(* Schneider Machine Expert - Basic project SEMÁFORO 1 VIA - SCHNEIDER ELECTRIC, file version 2.8.0.0 *)
(* ProjectInformations: Name=SEMAFORO 1 VIA, Description=Semáforo de 1 via com temporizadores., botão [LIGA], botão [DESLIGA] e repetição automática de ciclo. *)
(* UserInformations: LastName=Gagliano, FirstName=Leonardo *)

HARDWARE
  Cpu 0: TM221C40T
  EthernetConfiguration: NetworkName=M221, IpAllocationMode=FixedAddress, IpAddress=0.0.0.0, SubnetMask=0.0.0.0
  SerialLineConfiguration: Baud=Baud19200, Parity=ParityEven, DataBits=DataBits8, StopBits=StopBits1, PhysicalMedium=PhysicalMediumRs485, TransmissionMode=TransmissionModeModbusRtu, SlaveId=1, Addressing=SlaveAddressing
  MastTask: UsePeriodScanMode=false, PeriodScan=100
  FastTask: Period=255
  CpuBehavior: StartingMode=StartAsPreviousState, AutoSaveRamOnEeprom=true, WatchdogPeriod=250

SYMBOLS  (address, symbol, comment, settings)
  %M0       DESLIGA
  %TM0        [Preset=7, Base=OneSecond]
  %TM1        [Preset=3, Base=OneSecond]
  %TM2        [Preset=5, Base=OneSecond]
  %I0.0     LIGA
  %Q0.0     LUZ_VERMELHA
  %Q0.1     LUZ_AMARELA
  %Q0.2     LUZ_VERDE

POU Novo POU
  (* SectionNumber=1 *)

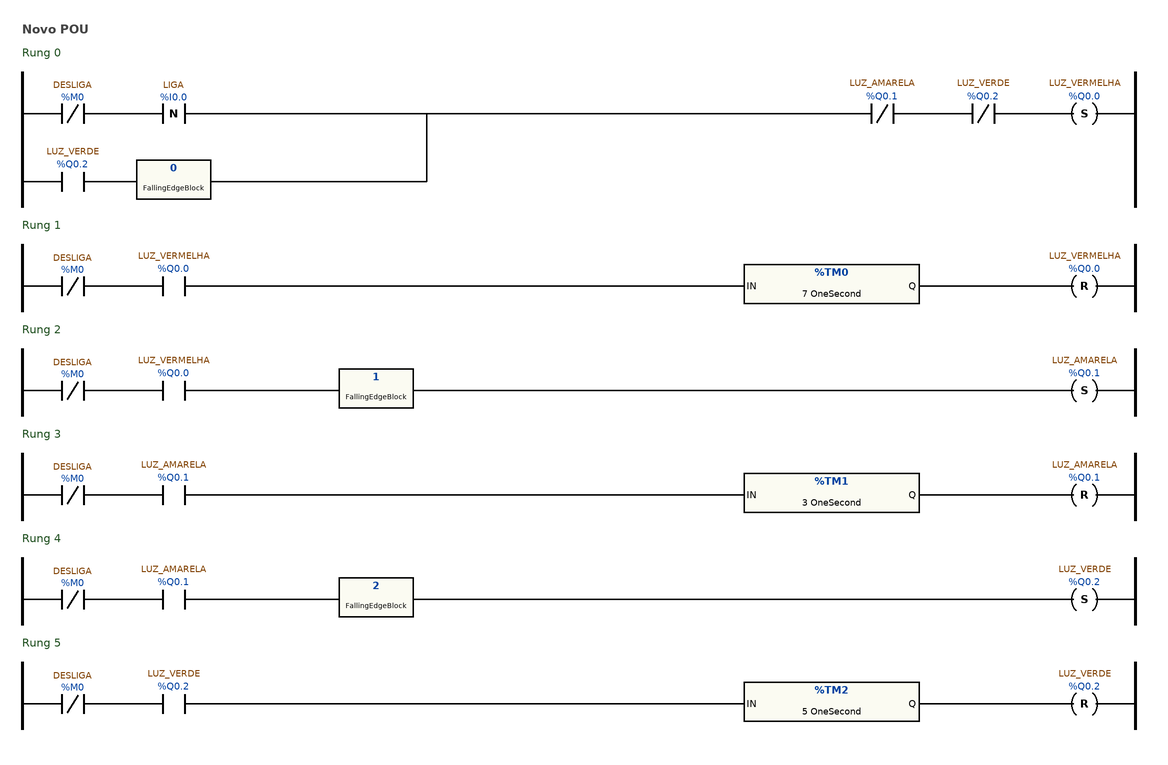

// Rung 0
  LDN %M0                 (* DESLIGA *)
  ANDF %I0.0              (* LIGA *)
  OR( %Q0.2               (* LUZ_VERDE *)
  FALLING0
  )
  ANDN %Q0.1              (* LUZ_AMARELA *)
  ANDN %Q0.2              (* LUZ_VERDE *)
  S %Q0.0                 (* LUZ_VERMELHA *)
  // as ST:
  //   IF (NOT DESLIGA AND FALLING(LIGA) OR FALLING(LUZ_VERDE)) AND NOT LUZ_AMARELA AND NOT LUZ_VERDE THEN LUZ_VERMELHA := TRUE; END_IF;

// Rung 1
  BLK %TM0
  LDN %M0                 (* DESLIGA *)
  AND %Q0.0               (* LUZ_VERMELHA *)
  IN
  OUT_BLK
  LD Q
  R %Q0.0                 (* LUZ_VERMELHA *)
  END_BLK
  // as ST:
  //   %TM0(IN := NOT DESLIGA AND LUZ_VERMELHA);
  //   IF %TM0.Q THEN LUZ_VERMELHA := FALSE; END_IF;

// Rung 2
  LDN %M0                 (* DESLIGA *)
  AND %Q0.0               (* LUZ_VERMELHA *)
  FALLING3
  S %Q0.1                 (* LUZ_AMARELA *)
  // as ST:
  //   IF FALLING(NOT DESLIGA AND LUZ_VERMELHA) THEN LUZ_AMARELA := TRUE; END_IF;

// Rung 3
  BLK %TM1
  LDN %M0                 (* DESLIGA *)
  AND %Q0.1               (* LUZ_AMARELA *)
  IN
  OUT_BLK
  LD Q
  R %Q0.1                 (* LUZ_AMARELA *)
  END_BLK
  // as ST:
  //   %TM1(IN := NOT DESLIGA AND LUZ_AMARELA);
  //   IF %TM1.Q THEN LUZ_AMARELA := FALSE; END_IF;

// Rung 4
  LDN %M0                 (* DESLIGA *)
  AND %Q0.1               (* LUZ_AMARELA *)
  FALLING2
  S %Q0.2                 (* LUZ_VERDE *)
  // as ST:
  //   IF FALLING(NOT DESLIGA AND LUZ_AMARELA) THEN LUZ_VERDE := TRUE; END_IF;

// Rung 5
  BLK %TM2
  LDN %M0                 (* DESLIGA *)
  AND %Q0.2               (* LUZ_VERDE *)
  IN
  OUT_BLK
  LD Q
  R %Q0.2                 (* LUZ_VERDE *)
  END_BLK
  // as ST:
  //   %TM2(IN := NOT DESLIGA AND LUZ_VERDE);
  //   IF %TM2.Q THEN LUZ_VERDE := FALSE; END_IF;
